{attribute addProperty BoxType "EJ2008-0000-0017"}
{attribute addProperty Id "ChannelAT %Q*ARRAY[0..7] OF Channel_7F374EB06480WcStateAT %I*WcState_64F6A8C6810InfoDataAT %I*InfoData_192954DE1620"}
{attribute addProperty CRC "976687666"}
{attribute addProperty SizeInBites "88"}
{attribute addProperty SizeInBytes "11"}
TYPE EJ2008_04E0E56B :
STRUCT
	{attribute addProperty Name "Channel"}
	Channel : ARRAY[0..7] OF Channel_7F374EB0;
	{attribute addProperty Name "WcState"}
	WcState : WcState_64F6A8C6;
	{attribute addProperty Name "InfoData"}
	InfoData : InfoData_192954DE;
END_STRUCT
END_TYPE

(* stored: Version 1.2.0.0, ProductVersion 3.1.4024.9
   DUT EJ2008_04E0E56B: Id {62cf6b7c-ddd3-4174-8edd-8f0573dbcfff} *)
